FUNCTION_BLOCK FB_PrintingBedSync
VAR_INPUT
	bErrorReset		: BOOL;
END_VAR
VAR_OUTPUT
	// Statusinformationen
	bError        	: BOOL;				// Fehler
    nErrorID      	: UDINT;
    sErrorMsg 		: STRING(80);
END_VAR
VAR
	// ADS-Kommunikation
    fbReadADS_AtTemp	: FB_ReadAdsSymByName;
	fbReadADS_ActTemp	: FB_ReadAdsSymByName;
	fbWriteADS_SetTemp	: FB_WriteAdsSymByName;

    // Konfiguration
    sRemoteNetID		: T_AmsNetId 	:= '172.16.6.70.1.1'; 	// Ziel-AMS-NetID
    sRemotePort 		: T_AmsPort		:= 856; 				// Hexapod PLC
	tTimeout			: TIME			:= T#5S;				// Zeit bis zu ADS Timeout
	
	// Temp
	nADSErrorID			: UDINT;
	bReadBusy_AtTemp	: BOOL;
	bReadBusy_ActTemp	: BOOL;
	bWriteBusy_SetTemp	: BOOL;
	bError_AtTemp		: BOOL;
	bError_ActTemp		: BOOL;
	bError_SetTemp		: BOOL;
END_VAR

IF NOT bError OR bErrorReset THEN
fbReadADS_AtTemp(
	bRead			:= NOT bReadBusy_AtTemp,
	sNetId			:= sRemoteNetID,
	nPort			:= sRemotePort,
	sVarName		:= 'GVL_PrintingBed.Druckbett_T_valid',
	nLen			:= SIZEOF(GVL_PrintingBed.PrintingBed.bAtTemp),
	nDestAddr		:= ADR(GVL_PrintingBed.PrintingBed.bAtTemp),
	tTimeout		:= tTimeout,
	eComMode		:= E_AdsComMode.eAdsComModeFastCom,
	bClearOnError	:= bErrorReset,
	bBusy			=> bReadBusy_AtTemp,
	bError			=> bError_AtTemp,
	nErrorId		=> nADSErrorID);

fbReadADS_ActTemp(
	bRead			:= NOT bReadBusy_ActTemp,
	sNetId			:= sRemoteNetID,
	nPort			:= sRemotePort,
	sVarName		:= 'GVL_PrintingBed.Druckbett_Tist',
	nLen			:= SIZEOF(GVL_PrintingBed.PrintingBed.fActualTemp),
	nDestAddr		:= ADR(GVL_PrintingBed.PrintingBed.fActualTemp),
	tTimeout		:= tTimeout,
	eComMode		:= E_AdsComMode.eAdsComModeFastCom,
	bClearOnError	:= bErrorReset,
	bBusy			=> bReadBusy_ActTemp,
	bError			=> bError_ActTemp,
	nErrorId		=> nADSErrorID);

fbWriteADS_SetTemp(
	bWrite			:= NOT bWriteBusy_SetTemp,
	sNetId			:= sRemoteNetID,
	nPort			:= sRemotePort,
	sVarName		:= 'GVL_PrintingBed.Druckbett_Tsoll',
	nLen			:= SIZEOF(GVL_PrintingBed.PrintingBed.fSetTemp),
	nSrcAddr		:= ADR(GVL_PrintingBed.PrintingBed.fSetTemp),
	tTimeout		:= tTimeout,
	eComMode		:= E_AdsComMode.eAdsComModeFastCom,
	bBusy			=> bWriteBusy_SetTemp,
	bError			=> bError_SetTemp,
	nErrorId		=> nADSErrorID);
END_IF

bError := bError_AtTemp OR bError_ActTemp OR bError_SetTemp;

IF bErrorReset AND NOT bError THEN
	bErrorReset := FALSE;
	nErrorID := 0;
	sErrorMsg := '';
END_IF

IF bError THEN
	nErrorID := 4000;
	sErrorMsg := CONCAT('ADS Fehler: ', TO_STRING(nADSErrorID));
END_IF

END_FUNCTION_BLOCK

(* stored: Version 1.1.0.1
   POU FB_PrintingBedSync: Id {e2408a13-d36e-4f00-bb95-a396dbbcb0b1}, SpecialFunc None *)
